DATA_BLOCK "楼层计数_DB"
{ S7_Optimized_Access := 'TRUE' }
VERSION : 0.1
NON_RETAIN
"楼层计数"

BEGIN

END_DATA_BLOCK

